TYPE PwmOutputChannel :
STRUCT
	{attribute addProperty Name "PWM output"}
	PWMoutput AT %Q* : UINT;
END_STRUCT
END_TYPE

(* stored: Version 1.1.0.1, ProductVersion 3.1.4024.9
   DUT PwmOutputChannel: Id {b4789e41-a7cf-08b6-2189-0966affcc27d} *)
